// LS Electric XG5000 project: 컨베이어벨트와 센서 제어_2
// PLC LSPLC
// module base 0 slot 0: 입출력 모듈:XBC-DR14E (DC 24V 입력 8점, 릴레이 출력 6점)

PROGRAM NewProgram (task: 스캔 프로그램)

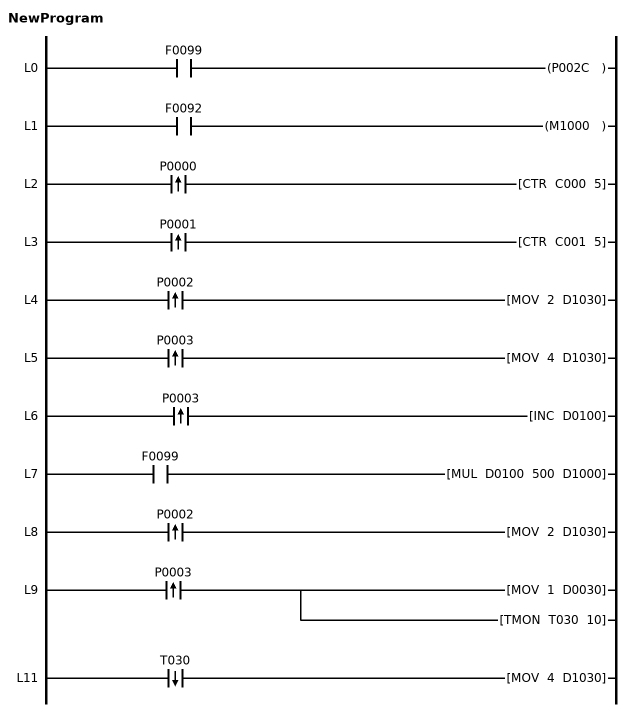
; L0
LOAD      F0099
OUT       P002C
; L1
LOAD      F0092
OUT       M1000
; L2
LOADP     P0000
CTR       C000 5
; L3
LOADP     P0001
CTR       C001 5
; L4
LOADP     P0002
MOV       2 D1030
; L5
LOADP     P0003
MOV       4 D1030
; L6
LOADP     P0003
INC       D0100
; L7
LOAD      F0099
MUL       D0100 500 D1000
; L8
LOADP     P0002
MOV       2 D1030
; L9
LOADP     P0003
MOV       1 D0030
TMON      T030 10
; L11
LOADN     T030
MOV       4 D1030